FUNCTION_BLOCK AutoResetIlck (* Basic Function Block Type *)
  (* Standard: 61499-2 *)
  (* Version 0.0, 8/3/2026, Schneider Electric, Template *)
  PACKAGE SE.Nereda;
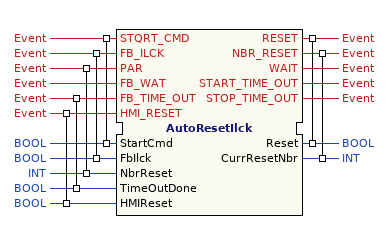
  EVENT_INPUT
    STQRT_CMD WITH StartCmd;
    FB_ILCK WITH FbIlck;
    PAR WITH NbrReset;
    FB_WAT;
    FB_TIME_OUT WITH TimeOutDone;
    HMI_RESET WITH HMIReset;
  END_EVENT
  EVENT_OUTPUT
    RESET WITH Reset;
    NBR_RESET WITH CurrResetNbr;
    WAIT;
    START_TIME_OUT;
    STOP_TIME_OUT;
  END_EVENT
  VAR_INPUT
    StartCmd : BOOL;
    FbIlck : BOOL;
    NbrReset : INT;
    TimeOutDone : BOOL;
    HMIReset : BOOL;
  END_VAR
  VAR_OUTPUT
    Reset : BOOL;
    CurrResetNbr : INT;
  END_VAR
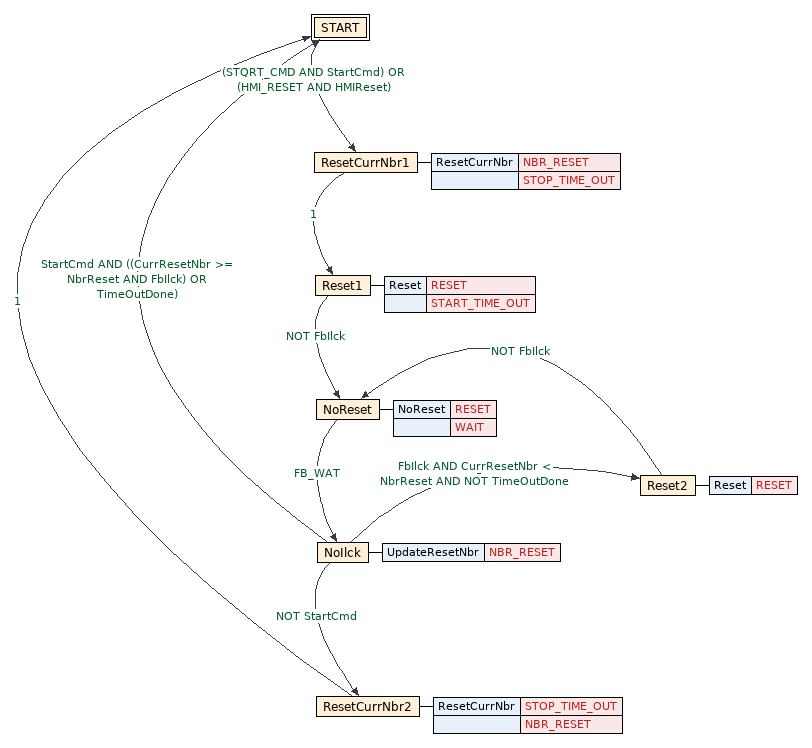
  EC_STATES
    START; (* Initial State *)
    Reset1 : Reset -> RESET, -> START_TIME_OUT;
    NoIlck : UpdateResetNbr -> NBR_RESET;
    Reset2 : Reset -> RESET;
    NoReset : NoReset -> RESET, -> WAIT;
    ResetCurrNbr2 : ResetCurrNbr -> STOP_TIME_OUT, -> NBR_RESET;
    ResetCurrNbr1 : ResetCurrNbr -> NBR_RESET, -> STOP_TIME_OUT;
  END_STATES
  EC_TRANSITIONS
    START TO ResetCurrNbr1 := (STQRT_CMD AND StartCmd) OR (HMI_RESET AND HMIReset);
    Reset1 TO NoReset := NOT FbIlck;
    NoIlck TO Reset2 := FbIlck AND CurrResetNbr < NbrReset AND NOT TimeOutDone;
    NoReset TO NoIlck := FB_WAT;
    Reset2 TO NoReset := NOT FbIlck;
    NoIlck TO START := StartCmd AND ((CurrResetNbr >= NbrReset AND FbIlck) OR TimeOutDone);
    NoIlck TO ResetCurrNbr2 := NOT StartCmd;
    ResetCurrNbr2 TO START := 1;
    ResetCurrNbr1 TO Reset1 := 1;
  END_TRANSITIONS
  ALGORITHM Reset IN ST:
;
Reset := TRUE;
  END_ALGORITHM
  ALGORITHM UpdateResetNbr IN ST:
;
CurrResetNbr := CurrResetNbr + 1;
  END_ALGORITHM
  ALGORITHM NoReset IN ST:
;
Reset := FALSE;
  END_ALGORITHM
  ALGORITHM ResetCurrNbr IN ST:
;
CurrResetNbr := 0;
  END_ALGORITHM
END_FUNCTION_BLOCK
